{attribute addProperty BoxType "KL6211-0022"}
{attribute addProperty Id "Channel_1Channel_B93188B300"}
{attribute addProperty CRC "2901387760"}
{attribute addProperty SizeInBites "0"}
{attribute addProperty SizeInBytes "0"}
TYPE KL_ACEFA9F0 :
STRUCT
	{attribute addProperty Name "Channel_1"}
	Channel_1 : Channel_B93188B3;
END_STRUCT
END_TYPE

(* stored: Version 1.2.0.0, ProductVersion 3.1.4024.9
   DUT KL_ACEFA9F0: Id {0edd8be3-285d-417a-a72a-8afe774d1179} *)
